TYPE "PosFbk_Encoder_Alr"
VERSION : 0.1
// Block: PosFbk_Encoder_Alr
   STRUCT
      CommFault : Bool;
      SensorFault : Bool;
      NoRef : Bool;
      Resolution : Bool;
   END_STRUCT;

END_TYPE
